(* PLC project robot6axis_cams, Dassault Systèmes ControlBuild 2024x *)
(* stored: creationDateTime 2023-10-04T11:04:00-01:00 *)

PROGRAM robot6axis_ctrled.robot6axis_cams
  VAR_INPUT
    profileNr : DINT := 0;
  END_VAR
  VAR_INPUT
    HomeCmd : BOOL := false;
    MoveVelCmd : BOOL := false;
    MoveAbsCmd : BOOL := false;
    MoveVel1ManualCmd : BOOL := false;
    MoveVel2ManualCmd : BOOL := false;
    MoveAbs1ManualCmd : BOOL := false;
    MoveAbs2ManualCmd : BOOL := false;
    StopCmd : BOOL := false;
    MovePosition : REAL := 0.0;
    MoveSpeed : REAL := 100.0;
    MoveAcceleration : REAL := 100.0;
    MoveDeceleration : REAL := 100.0;
    offsetAxToMa : REAL := 0.0;
  END_VAR
  VAR_INPUT
    name1 : STRING(50) := 'CamAxis1_100.txt';
    name2 : STRING(50) := 'CamAxis2_100.txt';
    name3 : STRING(50) := 'CamAxis3_100.txt';
    name4 : STRING(50) := 'CamAxis4_100.txt';
    name5 : STRING(50) := 'CamAxis5_100.txt';
    name6 : STRING(50) := 'CamAxis6_100.txt';
    name1_rej : STRING(50) := 'CamAxis1_rej.txt';
    name2_rej : STRING(50) := 'CamAxis2_rej.txt';
    name3_rej : STRING(50) := 'CamAxis3_rej.txt';
    name4_rej : STRING(50) := 'CamAxis4_rej.txt';
    name5_rej : STRING(50) := 'CamAxis5_rej.txt';
    name6_rej : STRING(50) := 'CamAxis6_rej.txt';
  END_VAR
  VAR_OUTPUT
    slavePosition1 : REAL := 0.0;
    slavePosition2 : REAL := 0.0;
    slavePosition3 : REAL := 0.0;
    slavePosition4 : REAL := 0.0;
    slavePosition5 : REAL := 0.0;
    slavePosition6 : REAL := 0.0;
    ActualPositionAx : REAL := 0.0;
    masterPosition : REAL := 0.0;
  END_VAR

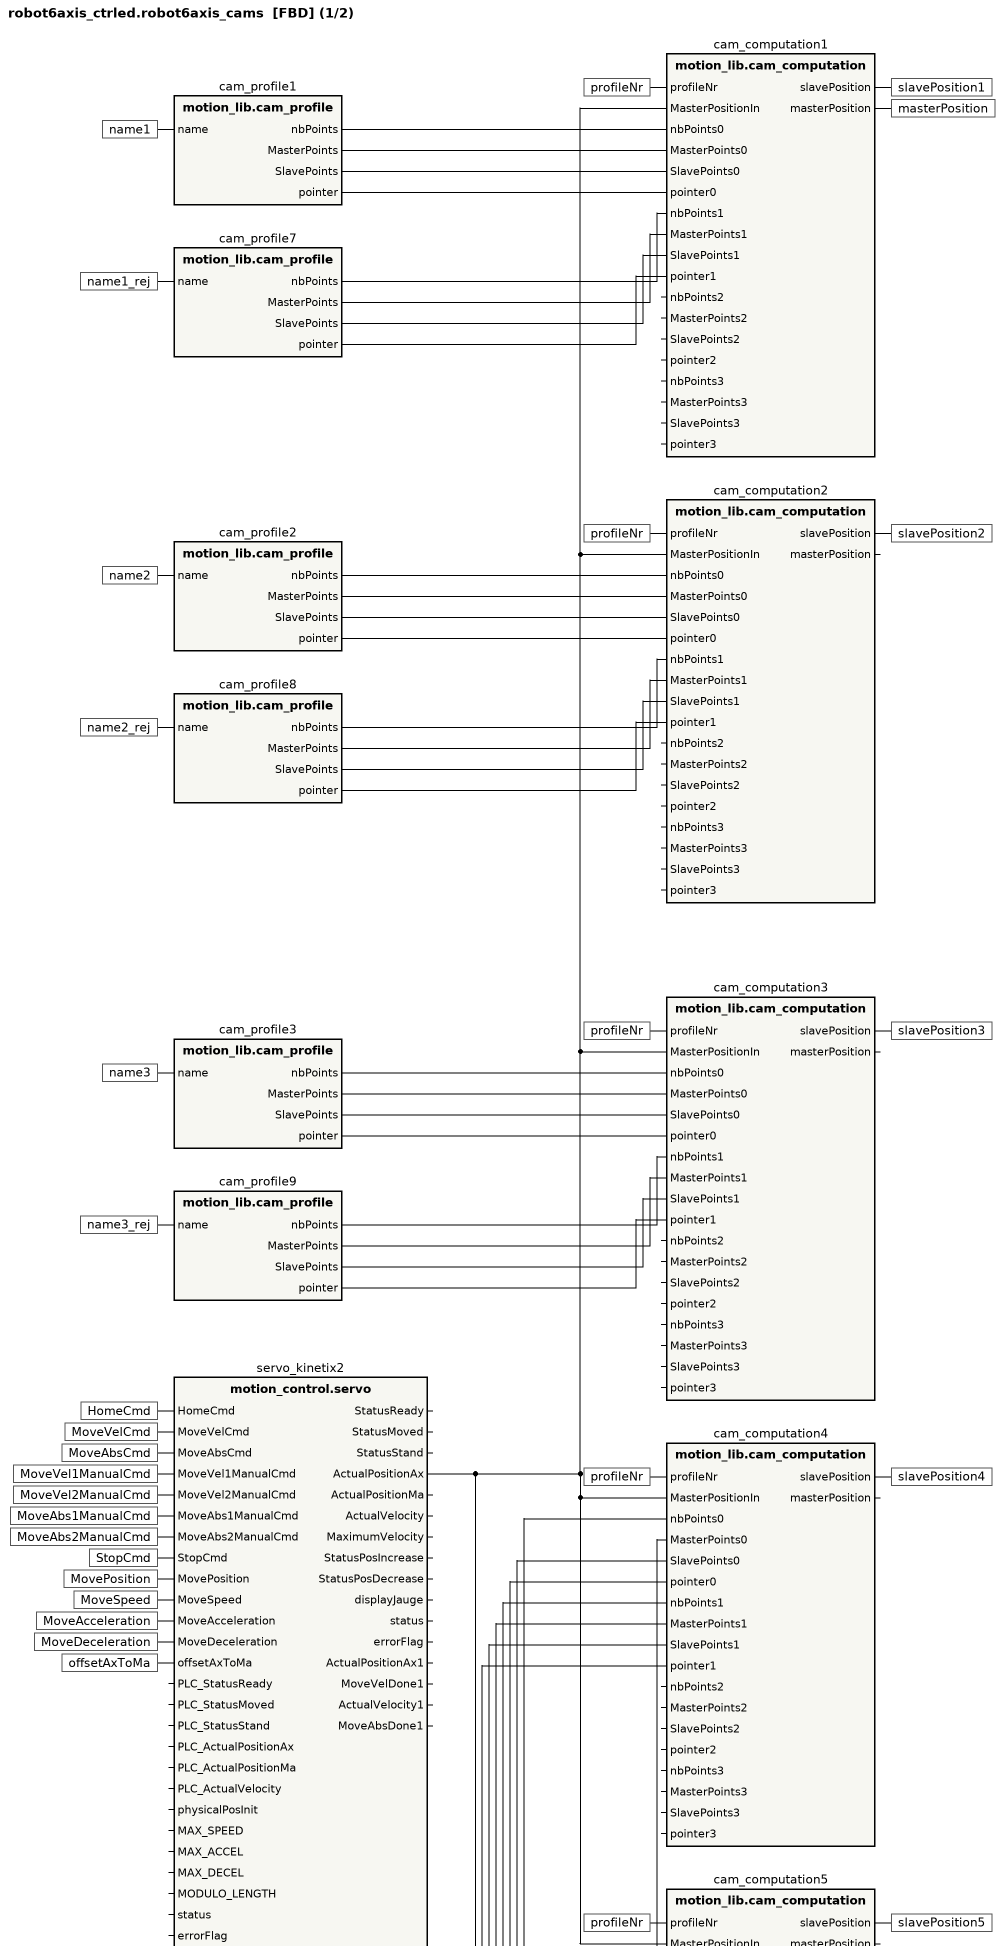
(* FBD diagram, written out as Structured Text *)
servo_kinetix2(HomeCmd := HomeCmd, MoveVelCmd := MoveVelCmd, MoveAbsCmd := MoveAbsCmd, MoveVel1ManualCmd := MoveVel1ManualCmd, MoveVel2ManualCmd := MoveVel2ManualCmd, MoveAbs1ManualCmd := MoveAbs1ManualCmd, MoveAbs2ManualCmd := MoveAbs2ManualCmd, StopCmd := StopCmd, MovePosition := MovePosition, MoveSpeed := MoveSpeed, MoveAcceleration := MoveAcceleration, MoveDeceleration := MoveDeceleration, offsetAxToMa := offsetAxToMa);
ActualPositionAx := servo_kinetix2.ActualPositionAx;
cam_profile1(name := name1);
cam_profile7(name := name1_rej);
cam_computation1(profileNr := profileNr, MasterPositionIn := servo_kinetix2.ActualPositionAx, nbPoints0 := cam_profile1.nbPoints, MasterPoints0 := cam_profile1.MasterPoints, SlavePoints0 := cam_profile1.SlavePoints, pointer0 := cam_profile1.pointer, nbPoints1 := cam_profile7.nbPoints, MasterPoints1 := cam_profile7.MasterPoints, SlavePoints1 := cam_profile7.SlavePoints, pointer1 := cam_profile7.pointer);
slavePosition1 := cam_computation1.slavePosition;
masterPosition := cam_computation1.masterPosition;
cam_profile2(name := name2);
cam_profile8(name := name2_rej);
cam_computation2(profileNr := profileNr, MasterPositionIn := servo_kinetix2.ActualPositionAx, nbPoints0 := cam_profile2.nbPoints, MasterPoints0 := cam_profile2.MasterPoints, SlavePoints0 := cam_profile2.SlavePoints, pointer0 := cam_profile2.pointer, nbPoints1 := cam_profile8.nbPoints, MasterPoints1 := cam_profile8.MasterPoints, SlavePoints1 := cam_profile8.SlavePoints, pointer1 := cam_profile8.pointer);
slavePosition2 := cam_computation2.slavePosition;
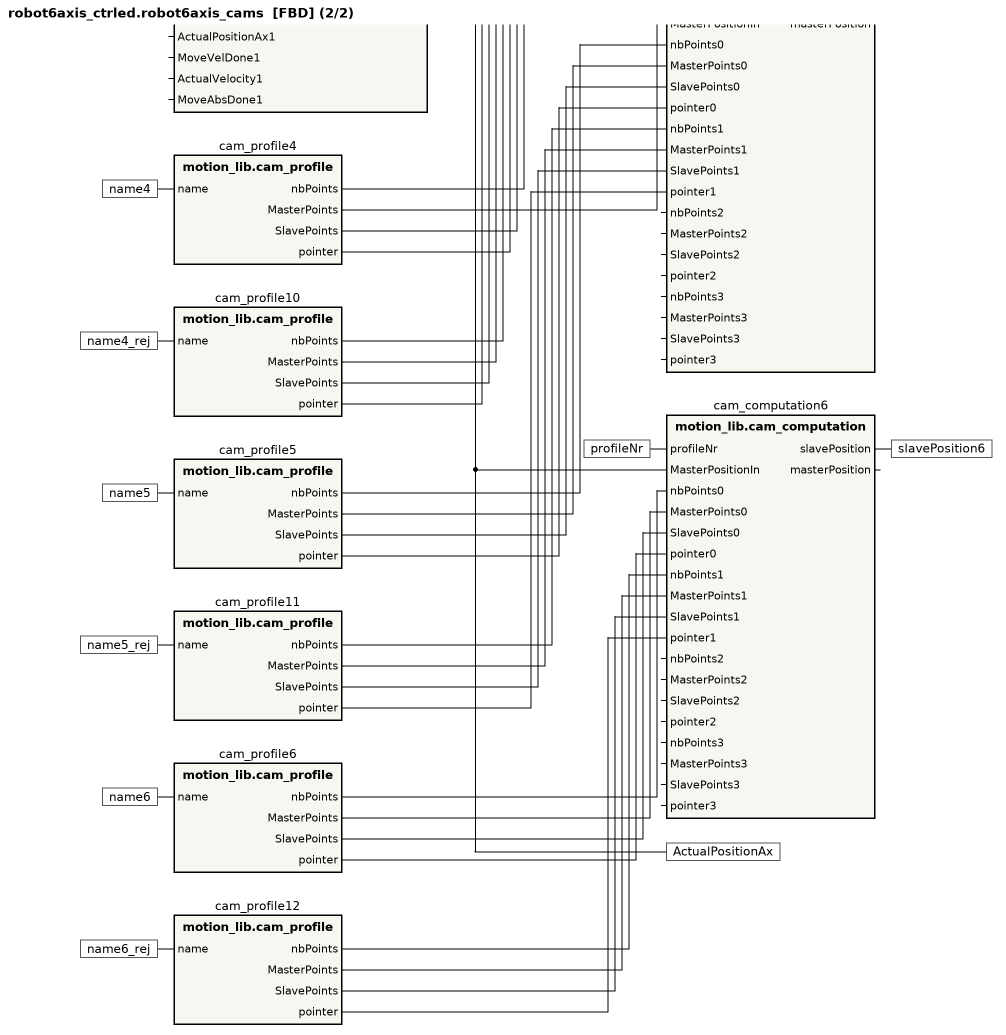
cam_profile3(name := name3);
cam_profile9(name := name3_rej);
cam_computation3(profileNr := profileNr, MasterPositionIn := servo_kinetix2.ActualPositionAx, nbPoints0 := cam_profile3.nbPoints, MasterPoints0 := cam_profile3.MasterPoints, SlavePoints0 := cam_profile3.SlavePoints, pointer0 := cam_profile3.pointer, nbPoints1 := cam_profile9.nbPoints, MasterPoints1 := cam_profile9.MasterPoints, SlavePoints1 := cam_profile9.SlavePoints, pointer1 := cam_profile9.pointer);
slavePosition3 := cam_computation3.slavePosition;
cam_profile4(name := name4);
cam_profile10(name := name4_rej);
cam_computation4(profileNr := profileNr, MasterPositionIn := servo_kinetix2.ActualPositionAx, nbPoints0 := cam_profile4.nbPoints, MasterPoints0 := cam_profile4.MasterPoints, SlavePoints0 := cam_profile4.SlavePoints, pointer0 := cam_profile4.pointer, nbPoints1 := cam_profile10.nbPoints, MasterPoints1 := cam_profile10.MasterPoints, SlavePoints1 := cam_profile10.SlavePoints, pointer1 := cam_profile10.pointer);
slavePosition4 := cam_computation4.slavePosition;
cam_profile5(name := name5);
cam_profile11(name := name5_rej);
cam_computation5(profileNr := profileNr, MasterPositionIn := servo_kinetix2.ActualPositionAx, nbPoints0 := cam_profile5.nbPoints, MasterPoints0 := cam_profile5.MasterPoints, SlavePoints0 := cam_profile5.SlavePoints, pointer0 := cam_profile5.pointer, nbPoints1 := cam_profile11.nbPoints, MasterPoints1 := cam_profile11.MasterPoints, SlavePoints1 := cam_profile11.SlavePoints, pointer1 := cam_profile11.pointer);
slavePosition5 := cam_computation5.slavePosition;
cam_profile6(name := name6);
cam_profile12(name := name6_rej);
cam_computation6(profileNr := profileNr, MasterPositionIn := servo_kinetix2.ActualPositionAx, nbPoints0 := cam_profile6.nbPoints, MasterPoints0 := cam_profile6.MasterPoints, SlavePoints0 := cam_profile6.SlavePoints, pointer0 := cam_profile6.pointer, nbPoints1 := cam_profile12.nbPoints, MasterPoints1 := cam_profile12.MasterPoints, SlavePoints1 := cam_profile12.SlavePoints, pointer1 := cam_profile12.pointer);
slavePosition6 := cam_computation6.slavePosition;
END_PROGRAM
